Staubli VAL3: save_AxisType.dtx

public num nValue
public string sName
